SUBAPPLICATION AuxInput_Licht_UP (* Subapplication Type *)
  (* Standard: 61499-2 *)
  (* Version 1.0, 2023-02-06, franz *)
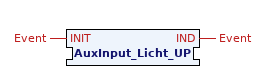
  EVENT_INPUT
    INIT;
  END_EVENT
  EVENT_OUTPUT
    IND;
  END_EVENT
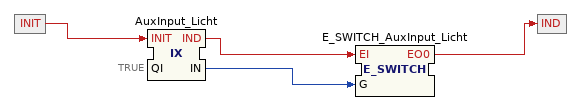
  FBS
    E_SWITCH_AuxInput_Licht : E_SWITCH;
    AuxInput_Licht : IX(QI := TRUE);
  END_FBS
  EVENT_CONNECTIONS
    AuxInput_Licht.IND TO E_SWITCH_AuxInput_Licht.EI;
    INIT TO AuxInput_Licht.INIT;
    E_SWITCH_AuxInput_Licht.EO0 TO IND;
  END_CONNECTIONS
  DATA_CONNECTIONS
    AuxInput_Licht.IN TO E_SWITCH_AuxInput_Licht.G;
  END_CONNECTIONS
END_SUBAPPLICATION
